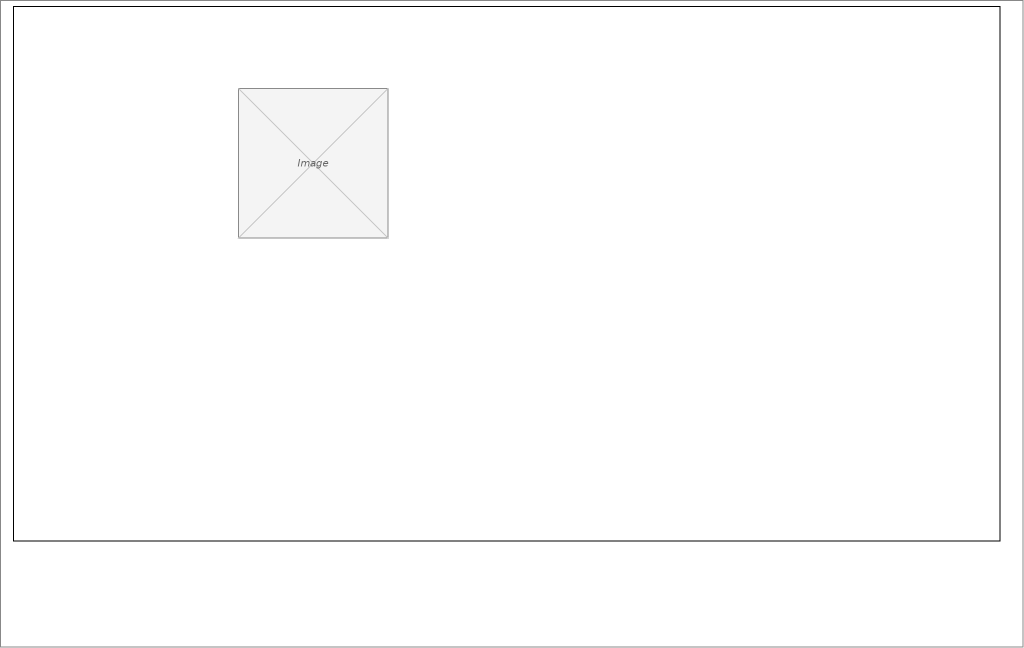
VISUALIZATION Statystyki  // 1024x648
    Rectangle (13,6 987x535)
    Image (238,88 150x150)
END_VISUALIZATION

(* stored: Version 1.1.0.1, ProductVersion 3.1.4022.10
   Visu Statystyki: Id {250b9449-0a93-42f0-ae83-4c8ccfad873a} *)
